PROGRAM MAIN
VAR
	safety	: FB_SafetyBase;	

	ax5_chA : FB_AxisBase;
	//ax8_chA : FB_AxisBase;
END_VAR

safety();
ax5_chA();
//ax8_chA();

END_PROGRAM

(* stored: Version 1.1.0.1, ProductVersion 3.1.4024.13
   POU MAIN: Id {a902c543-c0d9-4b6a-9ace-3646a5f5408f}, SpecialFunc None *)
